// TIA Portal V18 export
// export: Created 2026-06-22T15:41:34.4637002Z, ExportSetting WithDefaults, DisplayName Totally Integrated Automation Portal, DisplayVersion V18, DisplayName TIA Portal Openness, DisplayVersion V18, DisplayName TIA Portal Version Control Interface, DisplayVersion V18, DisplayName STEP 7 Professional, DisplayVersion V18, DisplayName STEP 7 Safety, DisplayVersion V18, DisplayName WinCC Professional, DisplayVersion V18
ORGANIZATION_BLOCK "Main"   // OB1, LAD, ProgramCycle
TITLE = "Main Program Sweep (Cycle)"
{ S7_Optimized_Access := 'TRUE' }
VERSION : 0.1
// stored: AutoNumber true, IsIECCheckEnabled false, SetENOAutomatically false
   VAR_INPUT
      Initial_Call : Bool;   // Initial call of this OB
      Remanence : Bool;   // =True, if remanent data are available
   END_VAR
BEGIN

REGION Network 1: Call FC_PLC2_Logic (Convert + Step Advance)
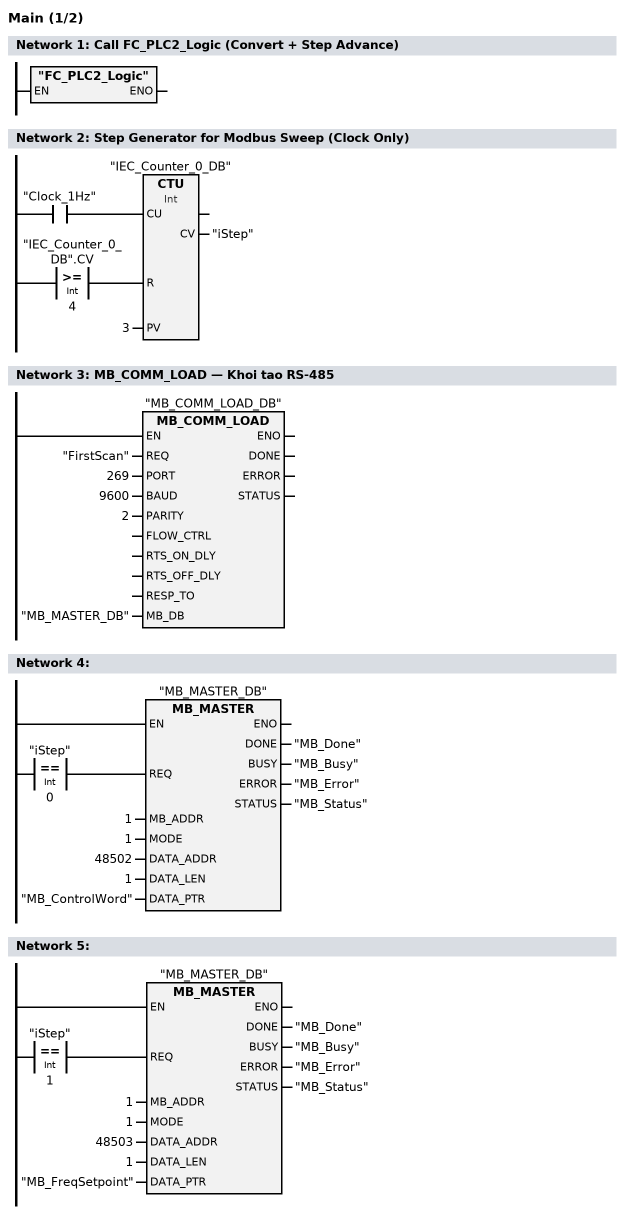
   RUNG wire#powerrail
      "FC_PLC2_Logic"()
   END_RUNG
   // the same network as SCL:
   "FC_PLC2_Logic"();
END_REGION

REGION Network 2: Step Generator for Modbus Sweep (Clock Only)
   RUNG wire#powerrail
      Contact( "Clock_1Hz" )
      { S7_Templates := "value_type := Int" } "IEC_Counter_0_DB".CTU(r := wire#w1, pv := 3, cv => "iStep")
   END_RUNG
   RUNG wire#powerrail
      { S7_Templates := "SrcType := Int" } GE_Contact(in1 := "IEC_Counter_0_DB".CV, in2 := 4)
   END_RUNG wire#w1
   // the same network as SCL:
   "IEC_Counter_0_DB".CTU(CU := "Clock_1Hz", R := "IEC_Counter_0_DB".CV >= 4, PV := 3, CV => "iStep");
END_REGION

REGION Network 3: MB_COMM_LOAD — Khoi tao RS-485
   RUNG wire#powerrail
      "MB_COMM_LOAD_DB".MB_COMM_LOAD(REQ := "FirstScan", PORT := 269, BAUD := 9600, PARITY := 2, FLOW_CTRL :=, RTS_ON_DLY :=, RTS_OFF_DLY :=, RESP_TO :=, MB_DB := "MB_MASTER_DB", DONE =>, ERROR =>, STATUS =>)
   END_RUNG
   // the same network as SCL:
   "MB_COMM_LOAD_DB"(REQ := "FirstScan", PORT := 269, BAUD := 9600, PARITY := 2, MB_DB := "MB_MASTER_DB");   // MB_COMM_LOAD
END_REGION

REGION Network 4
   RUNG wire#powerrail
      "MB_MASTER_DB".MB_MASTER(REQ := wire#w1, MB_ADDR := 1, MODE := 1, DATA_ADDR := 48502, DATA_LEN := 1, DATA_PTR := "MB_ControlWord", DONE => "MB_Done", BUSY => "MB_Busy", ERROR => "MB_Error", STATUS => "MB_Status")
   END_RUNG
   RUNG wire#powerrail
      { S7_Templates := "SrcType := Int" } EQ_Contact(in1 := "iStep", in2 := 0)
   END_RUNG wire#w1
   // the same network as SCL:
   "MB_MASTER_DB"(REQ := "iStep" = 0,   // MB_MASTER
                  MB_ADDR := 1,
                  MODE := 1,
                  DATA_ADDR := 48502,
                  DATA_LEN := 1,
                  DATA_PTR := "MB_ControlWord",
                  DONE => "MB_Done",
                  BUSY => "MB_Busy",
                  ERROR => "MB_Error",
                  STATUS => "MB_Status");
END_REGION

REGION Network 5
   RUNG wire#powerrail
      "MB_MASTER_DB".MB_MASTER(REQ := wire#w1, MB_ADDR := 1, MODE := 1, DATA_ADDR := 48503, DATA_LEN := 1, DATA_PTR := "MB_FreqSetpoint", DONE => "MB_Done", BUSY => "MB_Busy", ERROR => "MB_Error", STATUS => "MB_Status")
   END_RUNG
   RUNG wire#powerrail
      { S7_Templates := "SrcType := Int" } EQ_Contact(in1 := "iStep", in2 := 1)
   END_RUNG wire#w1
   // the same network as SCL:
   "MB_MASTER_DB"(REQ := "iStep" = 1,   // MB_MASTER
                  MB_ADDR := 1,
                  MODE := 1,
                  DATA_ADDR := 48503,
                  DATA_LEN := 1,
                  DATA_PTR := "MB_FreqSetpoint",
                  DONE => "MB_Done",
                  BUSY => "MB_Busy",
                  ERROR => "MB_Error",
                  STATUS => "MB_Status");
END_REGION

REGION Network 6
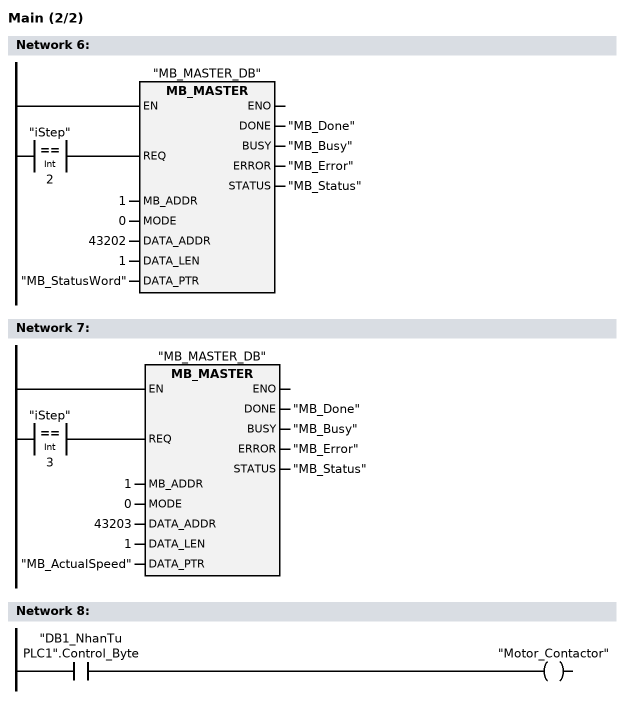
   RUNG wire#powerrail
      "MB_MASTER_DB".MB_MASTER(REQ := wire#w1, MB_ADDR := 1, MODE := 0, DATA_ADDR := 43202, DATA_LEN := 1, DATA_PTR := "MB_StatusWord", DONE => "MB_Done", BUSY => "MB_Busy", ERROR => "MB_Error", STATUS => "MB_Status")
   END_RUNG
   RUNG wire#powerrail
      { S7_Templates := "SrcType := Int" } EQ_Contact(in1 := "iStep", in2 := 2)
   END_RUNG wire#w1
   // the same network as SCL:
   "MB_MASTER_DB"(REQ := "iStep" = 2,   // MB_MASTER
                  MB_ADDR := 1,
                  MODE := 0,
                  DATA_ADDR := 43202,
                  DATA_LEN := 1,
                  DATA_PTR := "MB_StatusWord",
                  DONE => "MB_Done",
                  BUSY => "MB_Busy",
                  ERROR => "MB_Error",
                  STATUS => "MB_Status");
END_REGION

REGION Network 7
   RUNG wire#powerrail
      "MB_MASTER_DB".MB_MASTER(REQ := wire#w1, MB_ADDR := 1, MODE := 0, DATA_ADDR := 43203, DATA_LEN := 1, DATA_PTR := "MB_ActualSpeed", DONE => "MB_Done", BUSY => "MB_Busy", ERROR => "MB_Error", STATUS => "MB_Status")
   END_RUNG
   RUNG wire#powerrail
      { S7_Templates := "SrcType := Int" } EQ_Contact(in1 := "iStep", in2 := 3)
   END_RUNG wire#w1
   // the same network as SCL:
   "MB_MASTER_DB"(REQ := "iStep" = 3,   // MB_MASTER
                  MB_ADDR := 1,
                  MODE := 0,
                  DATA_ADDR := 43203,
                  DATA_LEN := 1,
                  DATA_PTR := "MB_ActualSpeed",
                  DONE => "MB_Done",
                  BUSY => "MB_Busy",
                  ERROR => "MB_Error",
                  STATUS => "MB_Status");
END_REGION

REGION Network 8
   RUNG wire#powerrail
      Contact( "DB1_NhanTuPLC1".Control_Byte )
      Coil( "Motor_Contactor" )
   END_RUNG
   // the same network as SCL:
   "Motor_Contactor" := "DB1_NhanTuPLC1".Control_Byte;
END_REGION
END_ORGANIZATION_BLOCK
